# EPICS substitutions: iocBoot/obsolete/ioc13idc/ipUnidig.substitutions
file "$(IPUNIDIG)/db/IpUnidigLi.db"
{
pattern
{P,       R,          PORT,       SCAN}
{13IDC:,  Unidig1Li,  Unidig1, "I/O Intr"}
{13IDC:,  Unidig2Li,  Unidig2, "I/O Intr"}
{13IDC:,  Unidig3Li,  Unidig3, "I/O Intr"}
}

file "$(IPUNIDIG)/db/IpUnidigBi.db"
{
pattern
{P,       R,          PORT,    MASK,        SCAN}
{13IDC:, Unidig1Bi0,  Unidig1, 0x000001, "I/O Intr"}
{13IDC:, Unidig1Bi1,  Unidig1, 0x000002, "I/O Intr"}
{13IDC:, Unidig1Bi2,  Unidig1, 0x000004, "I/O Intr"}
{13IDC:, Unidig1Bi3,  Unidig1, 0x000008, "I/O Intr"}
{13IDC:, Unidig1Bi4,  Unidig1, 0x000010, "I/O Intr"}
{13IDC:, Unidig1Bi5,  Unidig1, 0x000020, "I/O Intr"}
{13IDC:, Unidig1Bi6,  Unidig1, 0x000040, "I/O Intr"}
{13IDC:, Unidig1Bi7,  Unidig1, 0x000080, "I/O Intr"}
{13IDC:, Unidig1Bi8,  Unidig1, 0x000100, "I/O Intr"}
{13IDC:, Unidig1Bi9,  Unidig1, 0x000200, "I/O Intr"}
{13IDC:, Unidig1Bi10, Unidig1, 0x000400, "I/O Intr"}
{13IDC:, Unidig1Bi11, Unidig1, 0x000800, "I/O Intr"}
{13IDC:, Unidig1Bi12, Unidig1, 0x001000, "I/O Intr"}
{13IDC:, Unidig1Bi13, Unidig1, 0x002000, "I/O Intr"}
{13IDC:, Unidig1Bi14, Unidig1, 0x004000, "I/O Intr"}
{13IDC:, Unidig1Bi15, Unidig1, 0x008000, "I/O Intr"}
{13IDC:, Unidig1Bi16, Unidig1, 0x010000, "I/O Intr"}
{13IDC:, Unidig1Bi17, Unidig1, 0x020000, "I/O Intr"}
{13IDC:, Unidig1Bi18, Unidig1, 0x040000, "I/O Intr"}
{13IDC:, Unidig1Bi19, Unidig1, 0x080000, "I/O Intr"}
{13IDC:, Unidig1Bi20, Unidig1, 0x100000, "I/O Intr"}
{13IDC:, Unidig1Bi21, Unidig1, 0x200000, "I/O Intr"}
{13IDC:, Unidig1Bi22, Unidig1, 0x400000, "I/O Intr"}
{13IDC:, Unidig1Bi23, Unidig1, 0x800000, "I/O Intr"}
{13IDC:, Unidig2Bi0,  Unidig2, 0x000001, "I/O Intr"}
{13IDC:, Unidig2Bi1,  Unidig2, 0x000002, "I/O Intr"}
{13IDC:, Unidig2Bi2,  Unidig2, 0x000004, "I/O Intr"}
{13IDC:, Unidig2Bi3,  Unidig2, 0x000008, "I/O Intr"}
{13IDC:, Unidig2Bi4,  Unidig2, 0x000010, "I/O Intr"}
{13IDC:, Unidig2Bi5,  Unidig2, 0x000020, "I/O Intr"}
{13IDC:, Unidig2Bi6,  Unidig2, 0x000040, "I/O Intr"}
{13IDC:, Unidig2Bi7,  Unidig2, 0x000080, "I/O Intr"}
{13IDC:, Unidig2Bi8,  Unidig2, 0x000100, "I/O Intr"}
{13IDC:, Unidig2Bi9,  Unidig2, 0x000200, "I/O Intr"}
{13IDC:, Unidig2Bi10, Unidig2, 0x000400, "I/O Intr"}
{13IDC:, Unidig2Bi11, Unidig2, 0x000800, "I/O Intr"}
{13IDC:, Unidig2Bi12, Unidig2, 0x001000, "I/O Intr"}
{13IDC:, Unidig2Bi13, Unidig2, 0x002000, "I/O Intr"}
{13IDC:, Unidig2Bi14, Unidig2, 0x004000, "I/O Intr"}
{13IDC:, Unidig2Bi15, Unidig2, 0x008000, "I/O Intr"}
{13IDC:, Unidig2Bi16, Unidig2, 0x010000, "I/O Intr"}
{13IDC:, Unidig2Bi17, Unidig2, 0x020000, "I/O Intr"}
{13IDC:, Unidig2Bi18, Unidig2, 0x040000, "I/O Intr"}
{13IDC:, Unidig2Bi19, Unidig2, 0x080000, "I/O Intr"}
{13IDC:, Unidig2Bi20, Unidig2, 0x100000, "I/O Intr"}
{13IDC:, Unidig2Bi21, Unidig2, 0x200000, "I/O Intr"}
{13IDC:, Unidig2Bi22, Unidig2, 0x400000, "I/O Intr"}
{13IDC:, Unidig2Bi23, Unidig2, 0x800000, "I/O Intr"}
{13IDC:, Unidig3Bi0,  Unidig3, 0x000001, "I/O Intr"}
{13IDC:, Unidig3Bi1,  Unidig3, 0x000002, "I/O Intr"}
{13IDC:, Unidig3Bi2,  Unidig3, 0x000004, "I/O Intr"}
{13IDC:, Unidig3Bi3,  Unidig3, 0x000008, "I/O Intr"}
{13IDC:, Unidig3Bi4,  Unidig3, 0x000010, "I/O Intr"}
{13IDC:, Unidig3Bi5,  Unidig3, 0x000020, "I/O Intr"}
{13IDC:, Unidig3Bi6,  Unidig3, 0x000040, "I/O Intr"}
{13IDC:, Unidig3Bi7,  Unidig3, 0x000080, "I/O Intr"}
{13IDC:, Unidig3Bi8,  Unidig3, 0x000100, "I/O Intr"}
{13IDC:, Unidig3Bi9,  Unidig3, 0x000200, "I/O Intr"}
{13IDC:, Unidig3Bi10, Unidig3, 0x000400, "I/O Intr"}
{13IDC:, Unidig3Bi11, Unidig3, 0x000800, "I/O Intr"}
{13IDC:, Unidig3Bi12, Unidig3, 0x001000, "I/O Intr"}
{13IDC:, Unidig3Bi13, Unidig3, 0x002000, "I/O Intr"}
{13IDC:, Unidig3Bi14, Unidig3, 0x004000, "I/O Intr"}
{13IDC:, Unidig3Bi15, Unidig3, 0x008000, "I/O Intr"}
{13IDC:, Unidig3Bi16, Unidig3, 0x010000, "I/O Intr"}
{13IDC:, Unidig3Bi17, Unidig3, 0x020000, "I/O Intr"}
{13IDC:, Unidig3Bi18, Unidig3, 0x040000, "I/O Intr"}
{13IDC:, Unidig3Bi19, Unidig3, 0x080000, "I/O Intr"}
{13IDC:, Unidig3Bi20, Unidig3, 0x100000, "I/O Intr"}
{13IDC:, Unidig3Bi21, Unidig3, 0x200000, "I/O Intr"}
{13IDC:, Unidig3Bi22, Unidig3, 0x400000, "I/O Intr"}
{13IDC:, Unidig3Bi23, Unidig3, 0x800000, "I/O Intr"}

}

file "$(IPUNIDIG)/db/IpUnidigBo.db"
{
pattern
{P,       R,        PORT,    MASK}
{13IDC:, Unidig1Bo0,  Unidig1, 0x000001}
{13IDC:, Unidig1Bo1,  Unidig1, 0x000002}
{13IDC:, Unidig1Bo2,  Unidig1, 0x000004}
{13IDC:, Unidig1Bo3,  Unidig1, 0x000008}
{13IDC:, Unidig1Bo4,  Unidig1, 0x000010}
{13IDC:, Unidig1Bo5,  Unidig1, 0x000020}
{13IDC:, Unidig1Bo6,  Unidig1, 0x000040}
{13IDC:, Unidig1Bo7,  Unidig1, 0x000080}
{13IDC:, Unidig1Bo8,  Unidig1, 0x000100}
{13IDC:, Unidig1Bo9,  Unidig1, 0x000200}
{13IDC:, Unidig1Bo10, Unidig1, 0x000400}
{13IDC:, Unidig1Bo11, Unidig1, 0x000800}
{13IDC:, Unidig1Bo12, Unidig1, 0x001000}
{13IDC:, Unidig1Bo13, Unidig1, 0x002000}
{13IDC:, Unidig1Bo14, Unidig1, 0x004000}
{13IDC:, Unidig1Bo15, Unidig1, 0x008000}
{13IDC:, Unidig1Bo16, Unidig1, 0x010000}
{13IDC:, Unidig1Bo17, Unidig1, 0x020000}
{13IDC:, Unidig1Bo18, Unidig1, 0x040000}
{13IDC:, Unidig1Bo19, Unidig1, 0x080000}
{13IDC:, Unidig1Bo20, Unidig1, 0x100000}
{13IDC:, Unidig1Bo21, Unidig1, 0x200000}
{13IDC:, Unidig1Bo22, Unidig1, 0x400000}
{13IDC:, Unidig1Bo23, Unidig1, 0x800000}
{13IDC:, Unidig2Bo0,  Unidig2, 0x000001}
{13IDC:, Unidig2Bo1,  Unidig2, 0x000002}
{13IDC:, Unidig2Bo2,  Unidig2, 0x000004}
{13IDC:, Unidig2Bo3,  Unidig2, 0x000008}
{13IDC:, Unidig2Bo4,  Unidig2, 0x000010}
{13IDC:, Unidig2Bo5,  Unidig2, 0x000020}
{13IDC:, Unidig2Bo6,  Unidig2, 0x000040}
{13IDC:, Unidig2Bo7,  Unidig2, 0x000080}
{13IDC:, Unidig2Bo8,  Unidig2, 0x000100}
{13IDC:, Unidig2Bo9,  Unidig2, 0x000200}
{13IDC:, Unidig2Bo10, Unidig2, 0x000400}
{13IDC:, Unidig2Bo11, Unidig2, 0x000800}
{13IDC:, Unidig2Bo12, Unidig2, 0x001000}
{13IDC:, Unidig2Bo13, Unidig2, 0x002000}
{13IDC:, Unidig2Bo14, Unidig2, 0x004000}
{13IDC:, Unidig2Bo15, Unidig2, 0x008000}
{13IDC:, Unidig2Bo16, Unidig2, 0x010000}
{13IDC:, Unidig2Bo17, Unidig2, 0x020000}
{13IDC:, Unidig2Bo18, Unidig2, 0x040000}
{13IDC:, Unidig2Bo19, Unidig2, 0x080000}
{13IDC:, Unidig2Bo20, Unidig2, 0x100000}
{13IDC:, Unidig2Bo21, Unidig2, 0x200000}
{13IDC:, Unidig2Bo22, Unidig2, 0x400000}
{13IDC:, Unidig2Bo23, Unidig2, 0x800000}
{13IDC:, Unidig3Bo0,  Unidig3, 0x000001}
{13IDC:, Unidig3Bo1,  Unidig3, 0x000002}
{13IDC:, Unidig3Bo2,  Unidig3, 0x000004}
{13IDC:, Unidig3Bo3,  Unidig3, 0x000008}
{13IDC:, Unidig3Bo4,  Unidig3, 0x000010}
{13IDC:, Unidig3Bo5,  Unidig3, 0x000020}
{13IDC:, Unidig3Bo6,  Unidig3, 0x000040}
{13IDC:, Unidig3Bo7,  Unidig3, 0x000080}
{13IDC:, Unidig3Bo8,  Unidig3, 0x000100}
{13IDC:, Unidig3Bo9,  Unidig3, 0x000200}
{13IDC:, Unidig3Bo10, Unidig3, 0x000400}
{13IDC:, Unidig3Bo11, Unidig3, 0x000800}
{13IDC:, Unidig3Bo12, Unidig3, 0x001000}
{13IDC:, Unidig3Bo13, Unidig3, 0x002000}
{13IDC:, Unidig3Bo14, Unidig3, 0x004000}
{13IDC:, Unidig3Bo15, Unidig3, 0x008000}
{13IDC:, Unidig3Bo16, Unidig3, 0x010000}
{13IDC:, Unidig3Bo17, Unidig3, 0x020000}
{13IDC:, Unidig3Bo18, Unidig3, 0x040000}
{13IDC:, Unidig3Bo19, Unidig3, 0x080000}
{13IDC:, Unidig3Bo20, Unidig3, 0x100000}
{13IDC:, Unidig3Bo21, Unidig3, 0x200000}
{13IDC:, Unidig3Bo22, Unidig3, 0x400000}
{13IDC:, Unidig3Bo23, Unidig3, 0x800000}
}

file "$(IPUNIDIG)/db/IpUnidigLo.db"
{
pattern
{P,       R,          PORT}
{13IDC:,  Unidig1Lo,  Unidig1}
{13IDC:,  Unidig2Lo,  Unidig2}
{13IDC:,  Unidig3Lo,  Unidig3}
}
